% RSLogix 500 project PUMP&VALVE-ANALOG.RSS, saved by version 8.30.00.16 %
PROJECT "UNTITLED"    % processor: Bul.1763 MicroLogix 1100 Series B %

PROGRAM FILES
  LAD 2 "MAIN"  4 rungs
  LAD 3 "I/O"  4 rungs
  LAD 4 "ALARMS"  7 rungs
  LAD 5 "CONTROLS"  5 rungs

DATA FILES
  O0 OUTPUT  12 elements
  I1 INPUT  10 elements
  S2 STATUS  66 elements
  B3 BINARY  2 elements
  T4 TIMER  4 elements
  C5 COUNTER  1 elements
  R6 CONTROL  1 elements
  N7 INTEGER  1 elements
  F8 FLOAT  1 elements

LADDER 2 "MAIN"
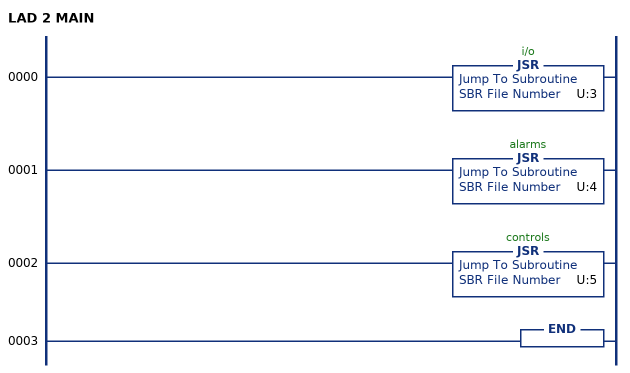
% Rung: 0 %
SOR JSR U:3 EOR
%   U:3  "i/o" %
% Rung: 1 %
SOR JSR U:4 EOR
%   U:4  "alarms" %
% Rung: 2 %
SOR JSR U:5 EOR
%   U:5  "controls" %
% Rung: 3 %
SOR END EOR

LADDER 3 "I/O"
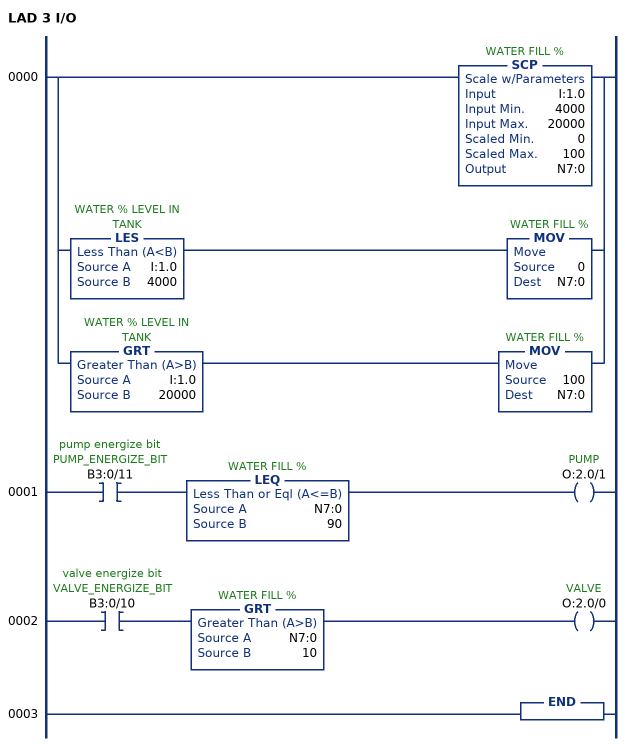
% Rung: 0 %
SOR BST SCP I:1.0 4000 20000 0 100 N7:0 NXB BST LES I:1.0 4000 MOV 0 N7:0 NXB GRT I:1.0 20000 MOV 100 N7:0 BND BND EOR
%   I:1.0  "WATER % LEVEL IN TANK" %
%   N7:0  "WATER FILL %" %
% Rung: 1 %
SOR XIC B3:0/11 LEQ N7:0 90 OTE O:2.0/1 EOR
%   B3:0/11  PUMP_ENERGIZE_BIT  "pump energize bit" %
%   N7:0  "WATER FILL %" %
%   O:2.0/1  "PUMP" %
% Rung: 2 %
SOR XIC B3:0/10 GRT N7:0 10 OTE O:2.0/0 EOR
%   B3:0/10  VALVE_ENERGIZE_BIT  "valve energize bit" %
%   N7:0  "WATER FILL %" %
%   O:2.0/0  "VALVE" %
% Rung: 3 %
SOR END EOR

LADDER 4 "ALARMS"
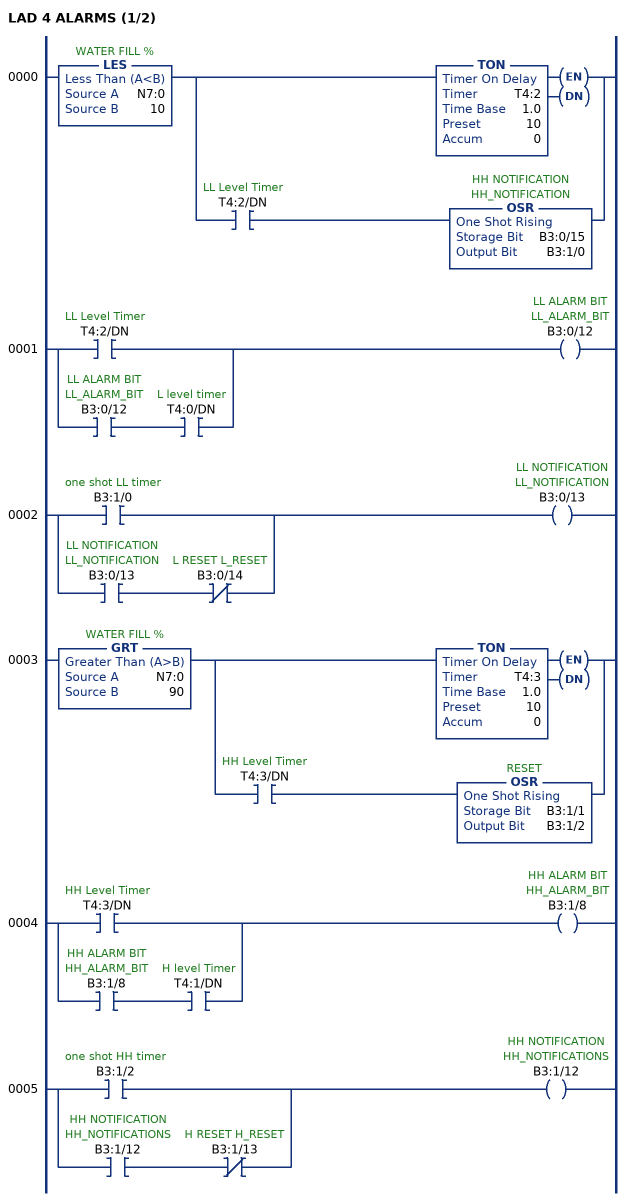
% Rung: 0 %
SOR LES N7:0 10 BST TON T4:2 1.0 10 0 NXB XIC T4:2/DN OSR B3:0/15 B3:1/0 BND EOR
%   N7:0  "WATER FILL %" %
%   T4:2/DN  "LL Level Timer" %
%   B3:0/15  HH_NOTIFICATION  "HH NOTIFICATION" %
%   B3:1/0  "one shot LL timer" %
% Rung: 1 %
SOR BST XIC T4:2/DN NXB XIC B3:0/12 XIC T4:0/DN BND OTE B3:0/12 EOR
%   T4:2/DN  "LL Level Timer" %
%   B3:0/12  LL_ALARM_BIT  "LL ALARM BIT" %
%   T4:0/DN  "L level timer" %
% Rung: 2 %
SOR BST XIC B3:1/0 NXB XIC B3:0/13 XIO B3:0/14 BND OTE B3:0/13 EOR
%   B3:1/0  "one shot LL timer" %
%   B3:0/13  LL_NOTIFICATION  "LL NOTIFICATION" %
%   B3:0/14  L_RESET  "L RESET" %
% Rung: 3 %
SOR GRT N7:0 90 BST TON T4:3 1.0 10 0 NXB XIC T4:3/DN OSR B3:1/1 B3:1/2 BND EOR
%   N7:0  "WATER FILL %" %
%   T4:3/DN  "HH Level Timer" %
%   B3:1/1  "RESET" %
%   B3:1/2  "one shot HH timer" %
% Rung: 4 %
SOR BST XIC T4:3/DN NXB XIC B3:1/8 XIC T4:1/DN BND OTE B3:1/8 EOR
%   T4:3/DN  "HH Level Timer" %
%   B3:1/8  HH_ALARM_BIT  "HH ALARM BIT" %
%   T4:1/DN  "H level Timer" %
% Rung: 5 %
SOR BST XIC B3:1/2 NXB XIC B3:1/12 XIO B3:1/13 BND OTE B3:1/12 EOR
%   B3:1/2  "one shot HH timer" %
%   B3:1/12  HH_NOTIFICATIONS  "HH NOTIFICATION" %
%   B3:1/13  H_RESET  "H RESET" %

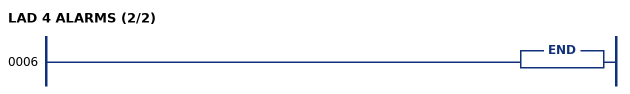
% Rung: 6 %
SOR END EOR

LADDER 5 "CONTROLS"
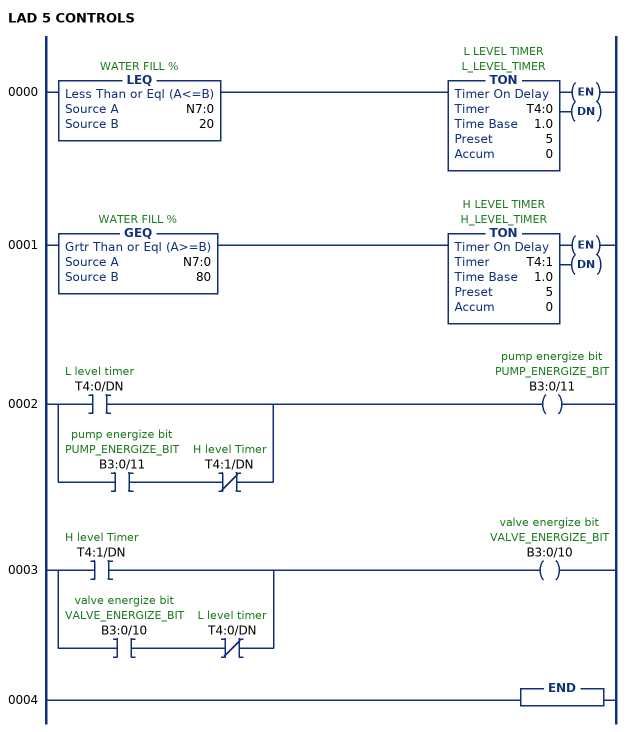
% Rung: 0 %
SOR LEQ N7:0 20 TON T4:0 1.0 5 0 EOR
%   N7:0  "WATER FILL %" %
%   T4:0  L_LEVEL_TIMER  "L LEVEL TIMER" %
% Rung: 1 %
SOR GEQ N7:0 80 TON T4:1 1.0 5 0 EOR
%   N7:0  "WATER FILL %" %
%   T4:1  H_LEVEL_TIMER  "H LEVEL TIMER" %
% Rung: 2 %
SOR BST XIC T4:0/DN NXB XIC B3:0/11 XIO T4:1/DN BND OTE B3:0/11 EOR
%   T4:0/DN  "L level timer" %
%   B3:0/11  PUMP_ENERGIZE_BIT  "pump energize bit" %
%   T4:1/DN  "H level Timer" %
% Rung: 3 %
SOR BST XIC T4:1/DN NXB XIC B3:0/10 XIO T4:0/DN BND OTE B3:0/10 EOR
%   T4:1/DN  "H level Timer" %
%   B3:0/10  VALVE_ENERGIZE_BIT  "valve energize bit" %
%   T4:0/DN  "L level timer" %
% Rung: 4 %
SOR END EOR

OTHER DOCUMENTED ADDRESSES
  B3:0/0  "L Level"
  B3:0/1  "H Level"
  B3:0/2  "LL Level"
  B3:0/3  "HH Level"
  B3:0/4  "valve"
  B3:0/5  "pump"
  B3:0/6  L_LEVEL_BIT  "L Level bit"
  B3:0/7  H_LEVEL_BIT  "H Level bit"
  B3:0/8  LL_LEVEL_BIT  "LL Level bit"
  B3:0/9  HH_LEVEL_BIT  "HH Level bit"
  B3:1/3  "LL ons bit"
  B3:1/4  "hh ons bit"
  B3:1/5  "HH NOTIFICATION"
  B3:1/6  "hh osr bit"
  B3:1/7  "ll osr bit"
  I:0.0/0  "L level switch"
  I:0.0/1  "H level switch"
  I:0.0/2  "LL level switch"
  I:0.0/3  "HH level switch"
  I:1.0/0  "L LEVEL SWTICH"
  I:1.0/1  "H LEVEL SWTICH"
  I:1.0/2  "LL LEVEL SWTICH"
  I:1.0/3  "HH LEVEL SWTICH"
  O:0.0/0  "valve"
  O:0.0/1  "pump"

DATA TABLE (non-zero values as saved)
DATA T4
% .PRE .ACC %
% T4:0 % 5 0
% T4:1 % 5 0
% T4:2 % 10 0
% T4:3 % 10 0
